// TwinCAT 3 PLC project lclsPLCMotionTest
// ProgramVersion: 3.1.4026.17
// libraries:
//   LCLS General, * (SLAC)
//   lcls-twincat-motion, * (SLAC)
//   PMPS, * (SLAC - LCLS)
//   Tc2_Standard, * (Beckhoff Automation GmbH)
//   Tc2_System, * (Beckhoff Automation GmbH)
// project tree:
//   DUTs/ ENUM_AxisStates.TcDUT, E_PMPSState.TcDUT
//   / PlcTask.TcTTO
//   POUs/ MAIN.TcPOU, STATES.TcPOU
// real-time tasks:
//   TASK PlcTask: cycle T#10ms, priority 20, ADS port 350
// motion (NC):
//   TASK NC-Task 1 SAF: cycle T#2ms, priority 4, ADS port 501
//   TASK NC-Task 1 SVB: cycle T#10ms, priority 8, ADS port 511
//   AXIS Axis_PMPS_M3 (id 3)
//     OtherSettings: AllowMotionCmdToSlave=true
//     encoder EncType=1
//       EncPara: ScaleFactorDenominator=2
//     drive DrvType=5
//       Analog: TorqueSetpointScale=10, ScaleFactorActTorque=0.1
//       TimeComp: TaskDelayCycles=1
//     controller CtrType=1
//       CtrPara: PriorControlFactor=1
//         Observer: BandWidth=20
//   AXIS Axis_PMPS_M2 (id 2)
//     OtherSettings: AllowMotionCmdToSlave=true
//     encoder EncType=1
//       EncPara: ScaleFactorDenominator=2
//     drive DrvType=5
//       Analog: TorqueSetpointScale=10, ScaleFactorActTorque=0.1
//       TimeComp: TaskDelayCycles=1
//     controller CtrType=1
//       CtrPara: PriorControlFactor=1
//         Observer: BandWidth=20
//   AXIS Axis_PMPS_M1 (id 1)
//     OtherSettings: AllowMotionCmdToSlave=true
//     encoder EncType=1
//       EncPara: ScaleFactorDenominator=2
//     drive DrvType=5
//       Analog: TorqueSetpointScale=10, ScaleFactorActTorque=0.1
//       TimeComp: TaskDelayCycles=1
//     controller CtrType=1
//       CtrPara: PriorControlFactor=1
//         Observer: BandWidth=20
// variable links:
//   motion_abstraction_sample Instance <-> NC-Task 1 SAF/Axes/Axis 1
//     PlcTask Inputs/GVL_Axes.Axes[1].NcToPlc <-> Outputs/ToPlc
//     PlcTask Outputs/GVL_Axes.Axes[1].PlcToNc <-> Inputs/FromPlc
//   motion_abstraction_sample Instance <-> NC-Task 1 SAF/Axes/Axis 2
//     PlcTask Inputs/GVL_Axes.Axes[2].NcToPlc <-> Outputs/ToPlc
//     PlcTask Outputs/GVL_Axes.Axes[2].PlcToNc <-> Inputs/FromPlc
//   motion_abstraction_sample Instance <-> NC-Task 1 SAF/Axes/Axis 3
//     PlcTask Inputs/GVL_Axes.Axes[3].NcToPlc <-> Outputs/ToPlc
//     PlcTask Outputs/GVL_Axes.Axes[3].PlcToNc <-> Inputs/FromPlc
//   motion_abstraction_sample Instance <-> NC-Task 1 SAF/Axes/Axis 4
//     PlcTask Inputs/GVL_Axes.Axes[4].NcToPlc <-> Outputs/ToPlc
//     PlcTask Outputs/GVL_Axes.Axes[4].PlcToNc <-> Inputs/FromPlc

CONFIGURATION lclsPLCMotionTest
    RESOURCE PLC ON TwinCAT3
        TASK PlcTask(INTERVAL := T#10ms, PRIORITY := 20);
        PROGRAM MAIN WITH PlcTask : MAIN;
    END_RESOURCE
END_CONFIGURATION

// ---- DUTs/ENUM_AxisStates.TcDUT
{attribute 'qualified_only'}
{attribute 'strict'}
{attribute 'to_string'}
TYPE ENUM_AxisStates :
(
    UNKNOWN := 0, // UNKNOWN must be in slot 0 or the FB breaks
    OUT := 1,
    YAG := 2,
    TT := 3
) UINT;
END_TYPE

// ---- DUTs/E_PMPSState.TcDUT
{attribute 'qualified_only'}
{attribute 'to_string'}
TYPE E_PMPSState :
(
        UNKNOWN:=0,
        OUT,
        TARGET1A,
        TARGET1B
)UINT;
END_TYPE

// ---- POUs/MAIN.TcPOU
PROGRAM MAIN
VAR
	(* Axis 1 *)
    {attribute 'pytmc' := 'pv: TST:MOTION:M1'}
    M1 : ST_MotionStage := (
        sName := 'TST:MOTION1',
        bPowerSelf := TRUE,
        nEnableMode := ENUM_StageEnableMode.DURING_MOTION,
        fHomePosition := 0.0,
        nHomingMode := ENUM_EpicsHomeCmd.NONE
    );
    fbMotionStage1 : FB_MotionStage;

    {attribute 'pytmc' := '
      pv: TST:MOTION:M1:STATES
      io: io
      expand: :%.2d
    '}
    astPositionState1 : ARRAY[1..GeneralConstants.MAX_STATES] OF ST_PositionState;

    (* Axis 2 *)
    {attribute 'pytmc' := 'pv: TST:MOTION:M2'}
    M2 : ST_MotionStage := (
        sName := 'TST:MOTION2',
        bPowerSelf := TRUE,
        nEnableMode := ENUM_StageEnableMode.DURING_MOTION,
        fHomePosition := 0.0,
        nHomingMode := ENUM_EpicsHomeCmd.NONE
    );
    fbMotionStage2 : FB_MotionStage;

    {attribute 'pytmc' := '
      pv: TST:MOTION:M2:STATES
      io: io
      expand: :%.2d
    '}
    astPositionState2 : ARRAY[1..GeneralConstants.MAX_STATES] OF ST_PositionState;

    (* Axis 3 *)
    {attribute 'pytmc' := 'pv: TST:MOTION:M3'}
    M3 : ST_MotionStage := (
        sName := 'TST:MOTION3',
        bPowerSelf := TRUE,
        nEnableMode := ENUM_StageEnableMode.DURING_MOTION,
        fHomePosition := 0.0,
        nHomingMode := ENUM_EpicsHomeCmd.NONE
    );
    fbMotionStage3 : FB_MotionStage;

    {attribute 'pytmc' := '
      pv: TST:MOTION:M3:STATES
      io: io
      expand: :%.2d
    '}
    astPositionState3 : ARRAY[1..GeneralConstants.MAX_STATES] OF ST_PositionState;

    {attribute 'pytmc' := '
      pv: TST:MOTION:STATES:SET
      io: io
    '}
    eSetPos : ENUM_AxisStates;

    {attribute 'pytmc' := '
      pv: TST:MOTION:STATES:GET
      io: i
    '}
    eGetPos : ENUM_AxisStates;
    fbFFHWO: FB_HardwareFFOutput;
    fbArbiter: FB_Arbiter(1);
	fbSubSysIO       	:  FB_DummyArbIO;
    fb_Move3D : FB_PositionStatePMPS3D;

    stDefault : ST_PositionState := (
        fDelta := 0.5,
        fVelocity := 25,
        bMoveOk := TRUE,
        bValid := TRUE
    );
	fbStateSetup : FB_StateSetupHelper;
    bLimitBackwardEnable1 : BOOL;
    bLimitBackwardEnable2 : BOOL;
    bLimitBackwardEnable3 : BOOL;
    bLimitForwardEnable1  : BOOL;
    bLimitForwardEnable2  : BOOL;
    bLimitForwardEnable3  : BOOL;
	bReadDBNow: BOOL;
	bEnableBeamParams : BOOL := TRUE;
END_VAR

MOTION_GVL.fbStandardPMPSDB(
    bEnable:=TRUE,
	sPlcName  := 'plc-tst-motion',
	sDirectory := '/home/ecs-user/pmpsdb/',
	io_fbFFHWO:=fbFFHWO
);

fbStateSetup(stPositionState := stDefault, bSetDefault := TRUE);

fbStateSetup(stPositionState := astPositionState1[E_PMPSState.OUT],      sName := 'OUT',         fPosition := 2.5);
astPositionState1[E_PMPSState.OUT].stPMPS.sPmpsState := 'TST:PF-OUT';
fbStateSetup(stPositionState := astPositionState1[E_PMPSState.TARGET1A], sName := 'TARGET1A',    fPosition := -8.54);
astPositionState1[E_PMPSState.TARGET1A].stPMPS.sPmpsState := 'TST:PF-TARGET1A';
fbStateSetup(stPositionState := astPositionState1[E_PMPSState.TARGET1B], sName := 'TARGET1B',    fPosition := 9.57);
astPositionState1[E_PMPSState.TARGET1B].stPMPS.sPmpsState := 'TST:PF-TARGET1B';

fbStateSetup(stPositionState := astPositionState2[E_PMPSState.OUT],      sName := 'OUT',         fPosition := 2.5);
astPositionState2[E_PMPSState.OUT].stPMPS.sPmpsState := 'TST:PF-OUT';
fbStateSetup(stPositionState := astPositionState2[E_PMPSState.TARGET1A], sName := 'TARGET1A',    fPosition := -8.54);
astPositionState2[E_PMPSState.TARGET1A].stPMPS.sPmpsState := 'TST:PF-TARGET1A';
fbStateSetup(stPositionState := astPositionState2[E_PMPSState.TARGET1B], sName := 'TARGET1B',    fPosition := 9.57);
astPositionState2[E_PMPSState.TARGET1B].stPMPS.sPmpsState := 'TST:PF-TARGET1B';

fbStateSetup(stPositionState := astPositionState3[E_PMPSState.OUT],      sName := 'OUT',         fPosition := 2.5);
astPositionState3[E_PMPSState.OUT].stPMPS.sPmpsState := 'TST:PF-OUT';
fbStateSetup(stPositionState := astPositionState3[E_PMPSState.TARGET1A], sName := 'TARGET1A',    fPosition := -8.54);
astPositionState3[E_PMPSState.TARGET1A].stPMPS.sPmpsState := 'TST:PF-TARGET1A';
fbStateSetup(stPositionState := astPositionState3[E_PMPSState.TARGET1B], sName := 'TARGET1B',    fPosition := 9.57);
astPositionState3[E_PMPSState.TARGET1B].stPMPS.sPmpsState := 'TST:PF-TARGET1B';

M1.bLimitForwardEnable  := bLimitForwardEnable1;
M1.bLimitBackwardEnable := bLimitBackwardEnable1;
M1.bHardwareEnable         := TRUE;
M2.bLimitForwardEnable  := bLimitForwardEnable2;
M2.bLimitBackwardEnable := bLimitBackwardEnable2;
M2.bHardwareEnable         := TRUE;

M3.bLimitForwardEnable  := bLimitForwardEnable3;
M3.bLimitBackwardEnable := bLimitBackwardEnable3;
M3.bHardwareEnable         := TRUE;

fbMotionStage1(stMotionStage := M1);
fbMotionStage2(stMotionStage := M2);
fbMotionStage3(stMotionStage := M3);

fb_Move3D(
    stMotionStage1    := M1,
    stMotionStage2    := M2,
    stMotionStage3    := M3,
    astPositionState1 := astPositionState1,
    astPositionState2 := astPositionState2,
    astPositionState3 := astPositionState3,
    eEnumSet          := eSetPos,
    eEnumGet          := eGetPos,
	sDeviceName		 := 'TST:PF',
	sTransitionKey	 := 'TST:PF-TRANSITION',
    fbFFHWO              := fbFFHWO,
    fbArbiter            := fbArbiter,
    bReadDBNow           := bReadDBNow,
    bEnableMotion        := TRUE,
    bEnableBeamParams    := bEnableBeamParams,
    bEnablePositionLimits:= TRUE
);

fbSubSysIO(LA := fbArbiter, FFO := fbFFHWO);
fbFFHWO.Execute();

END_PROGRAM

// ---- POUs/STATES.TcPOU
PROGRAM STATES
VAR
	(* Axis 1 *)
    {attribute 'pytmc' := 'pv: TST:MOTION:M1'}
    M1 : ST_MotionStage := (
        sName := 'TST:MOTION1',
        bPowerSelf := TRUE,
        nEnableMode := ENUM_StageEnableMode.DURING_MOTION,
        fHomePosition := 0.0,
        nHomingMode := ENUM_EpicsHomeCmd.NONE
    );
    fbMotionStage1 : FB_MotionStage;

    {attribute 'pytmc' := '
      pv: TST:MOTION:M1:STATES
      io: io
      expand: :%.2d
    '}
    astPositionState1 : ARRAY[1..GeneralConstants.MAX_STATES] OF ST_PositionState;

    (* Axis 2 *)
    {attribute 'pytmc' := 'pv: TST:MOTION:M2'}
    M2 : ST_MotionStage := (
        sName := 'TST:MOTION2',
        bPowerSelf := TRUE,
        nEnableMode := ENUM_StageEnableMode.DURING_MOTION,
        fHomePosition := 0.0,
        nHomingMode := ENUM_EpicsHomeCmd.NONE
    );
    fbMotionStage2 : FB_MotionStage;

    {attribute 'pytmc' := '
      pv: TST:MOTION:M2:STATES
      io: io
      expand: :%.2d
    '}
    astPositionState2 : ARRAY[1..GeneralConstants.MAX_STATES] OF ST_PositionState;

    (* Axis 3 *)
    {attribute 'pytmc' := 'pv: TST:MOTION:M3'}
    M3 : ST_MotionStage := (
        sName := 'TST:MOTION3',
        bPowerSelf := TRUE,
        nEnableMode := ENUM_StageEnableMode.DURING_MOTION,
        fHomePosition := 0.0,
        nHomingMode := ENUM_EpicsHomeCmd.NONE
    );
    fbMotionStage3 : FB_MotionStage;

    {attribute 'pytmc' := '
      pv: TST:MOTION:M3:STATES
      io: io
      expand: :%.2d
    '}
    astPositionState3 : ARRAY[1..GeneralConstants.MAX_STATES] OF ST_PositionState;

    {attribute 'pytmc' := '
      pv: TST:MOTION:STATES:SET
      io: io
    '}
    eSetPos : ENUM_AxisStates;

    {attribute 'pytmc' := '
      pv: TST:MOTION:STATES:GET
      io: i
    '}
    eGetPos : ENUM_AxisStates;

    fb_Move3D : FB_PositionState3D;

    stDefault : ST_PositionState := (
        fDelta := 0.5,
        fVelocity := 25,
        bMoveOk := TRUE,
        bValid := TRUE
    );
	fbStateSetup : FB_StateSetupHelper;
    bLimitBackwardEnable1 : BOOL;
    bLimitBackwardEnable2 : BOOL;
    bLimitBackwardEnable3 : BOOL;
    bLimitForwardEnable1  : BOOL;
    bLimitForwardEnable2  : BOOL;
    bLimitForwardEnable3  : BOOL;
END_VAR

(* ===== State setup — all axes, all states ===== *)
fbStateSetup(stPositionState := stDefault, bSetDefault := TRUE);
fbStateSetup(stPositionState := astPositionState1[1], sName := 'OUT', fPosition := 100.0);
fbStateSetup(stPositionState := astPositionState1[2], sName := 'YAG', fPosition := 200.0);
fbStateSetup(stPositionState := astPositionState1[3], sName := 'TT',  fPosition := 300.0);

fbStateSetup(stPositionState := astPositionState2[1], sName := 'OUT', fPosition := 100.0);
fbStateSetup(stPositionState := astPositionState2[2], sName := 'YAG', fPosition := 200.0);
fbStateSetup(stPositionState := astPositionState2[3], sName := 'TT',  fPosition := 300.0);

fbStateSetup(stPositionState := astPositionState3[1], sName := 'OUT', fPosition := 100.0);
fbStateSetup(stPositionState := astPositionState3[2], sName := 'YAG', fPosition := 200.0);
fbStateSetup(stPositionState := astPositionState3[3], sName := 'TT',  fPosition := 300.0);

(* ===== Limit enable wiring ===== *)
M1.bLimitForwardEnable  := bLimitForwardEnable1;
M1.bLimitBackwardEnable := bLimitBackwardEnable1;
M1.bHardwareEnable         := TRUE;
M2.bLimitForwardEnable  := bLimitForwardEnable2;
M2.bLimitBackwardEnable := bLimitBackwardEnable2;
M2.bHardwareEnable         := TRUE;

M3.bLimitForwardEnable  := bLimitForwardEnable3;
M3.bLimitBackwardEnable := bLimitBackwardEnable3;
M3.bHardwareEnable         := TRUE;
(* ===== Motion stage cyclic calls ===== *)
fbMotionStage1(stMotionStage := M1);
fbMotionStage2(stMotionStage := M2);
fbMotionStage3(stMotionStage := M3);

(* ===== 3D state mover ===== *)
fb_Move3D(
    stMotionStage1    := M1,
    stMotionStage2    := M2,
    stMotionStage3    := M3,
    astPositionState1 := astPositionState1,
    astPositionState2 := astPositionState2,
    astPositionState3 := astPositionState3,
    eEnumSet          := eSetPos,
    eEnumGet          := eGetPos,
    bEnable           := TRUE
);

END_PROGRAM
